PROGRAM MAIN
VAR
END_VAR

END_PROGRAM

(* stored: Version 1.1.0.1
   POU MAIN: Id {40a29346-b9ff-4067-855e-fa294bfdfdf9} *)
